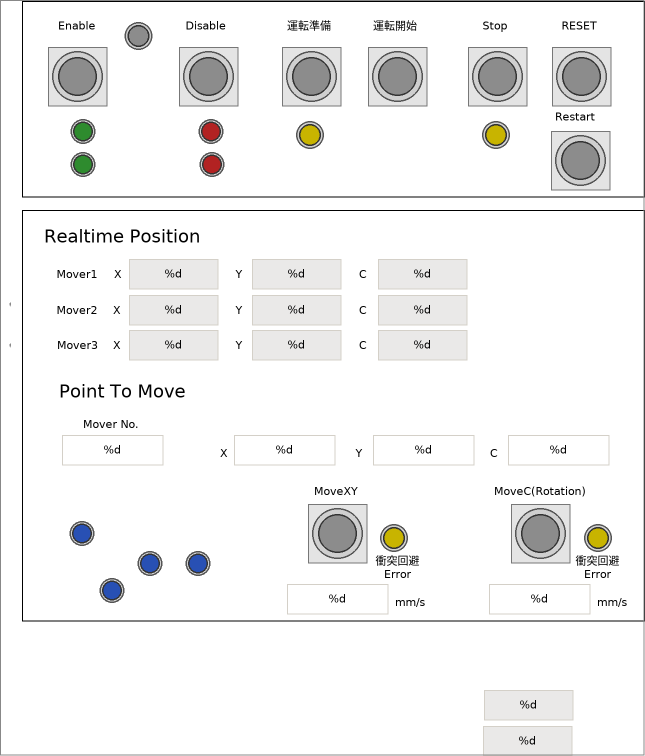
VISUALIZATION Visualization  // 645x756
    RoundedRectangle (22,1 623x196)
    RoundedRectangle (22,210 623x411)
    RockerSwitch (10,302 0x4), behaviour: TOGGLE, style: Switch-RockerSwitch-Gray
    PushSwitch (46,47 63x59), variable: MAIN.exeXpEnableMover, behaviour: TOGGLE, style: Switch-PushSwitch-Gray
    PushSwitch (177,47 63x59), variable: MAIN.exeXpDisableMover, behaviour: TOGGLE, style: Switch-PushSwitch-Gray
    Label (43,15 68x22), "Enable"
    Label (172,15 68x22), "Disable"
    Label (275,15 68x22), "運転準備"
    Label (541,106 68x22), "Restart"
    PushSwitch (280,47 63x59), variable: MAIN.exePreStartPB, behaviour: TOGGLE, style: Switch-PushSwitch-Gray
    PushSwitch (549,131 63x59), variable: MAIN.exerestartPB, behaviour: TOGGLE, style: Switch-PushSwitch-Gray
    PushSwitch (306,504 63x59), variable: MAIN.exeMoveXY, behaviour: TOGGLE, style: Switch-PushSwitch-Gray
    Textfield (234,435 101x30), "%d", text variable: MAIN.nManualX
        OnMouseClick: write the text variable via Default
    Textfield (373,435 101x30), "%d", text variable: MAIN.nManualY
        OnMouseClick: write the text variable via Default
    Textfield (508,435 101x30), "%d", text variable: MAIN.nManualC
        OnMouseClick: write the text variable via Default
    Label (168,442 112x23), "X"
    Label (303,442 112x23), "Y"
    Label (438,442 112x23), "C"
    Label (280,480 112x23), "MoveXY"
    Label (484,480 112x23), "MoveC(Rotation)"
    PushSwitch (509,504 63x59), variable: MAIN.exeMoveC, behaviour: TOGGLE, style: Switch-PushSwitch-Gray
    Textfield (62,435 101x30), "%d", text variable: MAIN.nMover
        OnMouseClick: write the text variable via Default
    Label (55,413 112x23), "Mover No."
    Lamp1 (378,519 32x38), variable: MAIN.ManualCollisionError[0], style: Lamp-Lamp1-Yellow
    Lamp1 (582,519 32x38), variable: MAIN.ManualCollisionError[1], style: Lamp-Lamp1-Yellow
    Lamp1 (294,116 32x38), variable: MAIN.bJoinDone, style: Lamp-Lamp1-Yellow
    Label (367,548 61x39), "衝突回避 Error"
    Label (567,548 61x39), "衝突回避 Error"
    Lamp1 (62,117 42x29), variable: MAIN.bMoverEnable[1], style: Lamp-Lamp1-Green
    Lamp1 (62,150 42x29), variable: MAIN.bMoverEnable[2], style: Lamp-Lamp1-Green
    Lamp1 (191,150 42x29), variable: MAIN.bMoverDisable[2], style: Lamp-Lamp1-Red
    Lamp1 (190,117 42x29), variable: MAIN.bMoverDisable[1], style: Lamp-Lamp1-Red
    PushSwitch (466,47 63x59), variable: MAIN.exeStop_os, behaviour: TOGGLE, style: Switch-PushSwitch-Gray
    Label (461,15 68x22), "Stop"
    Textfield (129,259 89x30), "%d", text variable: MAIN.VisVar[1][0]
    Textfield (252,259 89x30), "%d", text variable: MAIN.VisVar[1][1]
    Textfield (484,690 89x30), "%d", text variable: MAIN.VisVar[1][2]
    Label (62,263 112x23), "X"
    Label (183,263 112x23), "Y"
    Label (307,263 112x23), "C"
    Label (61,299 112x23), "X"
    Textfield (252,295 89x30), "%d", text variable: MAIN.VisVar[2][1]
    Textfield (483,726 89x30), "%d", text variable: MAIN.VisVar[2][2]
    Label (183,299 112x23), "Y"
    Label (307,299 112x23), "C"
    Textfield (129,295 89x30), "%d", text variable: MAIN.VisVar[2][0]
    Label (36,225 173x23), "Realtime Position"
    Label (21,263 112x23), "Mover1"
    Label (21,299 112x23), "Mover2"
    Label (36,380 173x23), "Point To Move"
    Textfield (489,584 101x30), "%d", text variable: MAIN.ValueC
        OnMouseClick: write the text variable via Default
    Label (545,15 68x22), "RESET"
    PushSwitch (550,47 63x59), variable: MAIN.exeresetPB, behaviour: TOGGLE, style: Switch-PushSwitch-Gray
    Textfield (378,259 89x30), "%d", text variable: MAIN.VisVar[1][3]
    Textfield (378,295 89x30), "%d", text variable: MAIN.VisVar[2][2]
    Textfield (287,584 101x30), "%d", text variable: MAIN.valueV
        OnMouseClick: write the text variable via Default
    Label (385,591 50x23), "mm/s"
    Label (587,591 50x23), "mm/s"
    Lamp1 (480,116 32x38), variable: MAIN.exeStop, style: Lamp-Lamp1-Yellow
    Lamp1 (121,20 35x32), variable: MAIN.fbAutoScan.bDone, style: Lamp-Lamp1-Gray
    RockerSwitch (10,343 0x4), behaviour: TOGGLE, style: Switch-RockerSwitch-Gray
    Label (61,334 112x23), "X"
    Label (183,334 112x23), "Y"
    Label (307,334 112x23), "C"
    Label (36,334 83x23), "Mover3"
    Textfield (129,330 89x30), "%d", text variable: MAIN.VisVar[3][0]
    Textfield (252,330 89x30), "%d", text variable: MAIN.VisVar[3][1]
    Textfield (378,330 89x30), "%d", text variable: MAIN.VisVar[3][2]
    Label (361,15 68x22), "運転開始"
    PushSwitch (366,47 63x59), variable: MAIN.exeStartPB, behaviour: TOGGLE, style: Switch-PushSwitch-Gray
    Lamp1 (91,576 42x29), variable: MAIN.StationBusy[1], style: Lamp-Lamp1-Blue
    Lamp1 (177,549 42x29), variable: MAIN.StationBusy[2], style: Lamp-Lamp1-Blue
    Lamp1 (129,549 42x29), variable: MAIN.StationBusy[3], style: Lamp-Lamp1-Blue
    Lamp1 (61,519 42x29), variable: MAIN.StationBusy[4], style: Lamp-Lamp1-Blue
END_VISUALIZATION

(* stored: Version 1.1.0.1
   Visu Visualization: Id {fe500f20-164b-4bed-a3cc-476b9fc24d00} *)
